{attribute 'linkalways'} 
{attribute 'no_explicit_call' := 'This FB is a CLASS and must be accessed using methods or properties'}
{attribute 'enable_dynamic_creation'}
FUNCTION_BLOCK Node_F_VN_CheckColorRange EXTENDS VisionNode
VAR
	ipSrcImage : _ITcVnImage;
    ipDestImage : _ITcVnImage;
    aLowerBounds : _TcVnVector4_LREAL;
    aUpperBounds : _TcVnVector4_LREAL;
    hrPrev : _HRESULT(S_OK);
	hresult : _HRESULT(S_OK);
END_VAR

METHOD PUBLIC  Clone : I_Node
VAR
	pNode : POINTER TO Node_F_VN_CheckColorRange;
END_VAR
pNode := __NEW(Node_F_VN_CheckColorRange);
Clone := pNode^;
END_METHOD

METHOD FB_init : BOOL
VAR_INPUT
	bInitRetains : BOOL; // if TRUE, the retain variables are initialized (warm start / cold start)
	bInCopyCode : BOOL;  // if TRUE, the instance afterwards gets moved into the copy code (online change)
END_VAR
AddInput('ipSrcImage', ipSrcImage);
AddInput('aLowerBounds', aLowerBounds);
AddInput('aUpperBounds', aUpperBounds);
AddInput('hrPrev', hrPrev);
AddOutput('ipDestImage', ipDestImage);
AddOutput('hresult', hresult);
END_METHOD

METHOD PROTECTED OnExecute
hresult.Value := F_VN_CheckColorRange(
	ipSrcImage := ipSrcImage.Value,
	ipDestImage := ipDestImage.Value,
    aLowerBounds := aLowerBounds.Value,
    aUpperBounds := aUpperBounds.Value,
	hrPrev := hrPrev.Value);
END_METHOD

METHOD PUBLIC PreExecutionCheck
VAR_INPUT
	Check : I_PreExecutionChecks;
END_VAR
Check.IsTrue(ipSrcImage.IsValid, 'ipSrcImage must contain an image');
END_METHOD

END_FUNCTION_BLOCK

(* stored: Version 1.1.0.1, ProductVersion 3.1.4024.15
   POU Node_F_VN_CheckColorRange: Id {6d4a5468-344d-0612-3e01-8256cacb09c4}, SpecialFunc None
   Folder Constructor: Id {4893eb66-04d1-0dd5-35ae-ff3355b8b059}
   Method Clone: Id {71df2436-1d2a-0a59-1ed9-bef283316911}
   Method FB_init: Id {657dc036-5751-0769-1d0b-090606cb1e7b}
   Method OnExecute: Id {f5a072fa-10be-0b9a-17da-87e9dc284840}
   Method PreExecutionCheck: Id {d073d69c-87ce-0568-139a-7c9b6ddbe930} *)
